// Mitsubishi GX Works2 project: 230927-005-nor   PLC: Q03UDV

// task Task_01 (event TRUE, interval 0, priority 31): POU_01

PROGRAM POU_01
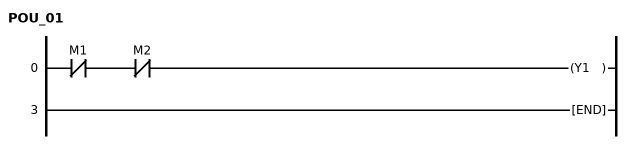
0     LDI     M1
      ANI     M2
      OUT     Y1
3     END
END_PROGRAM
